// Mitsubishi GX Works2 project: FRA 451 Class Project   PLC: FX3G

PROGRAM MAIN
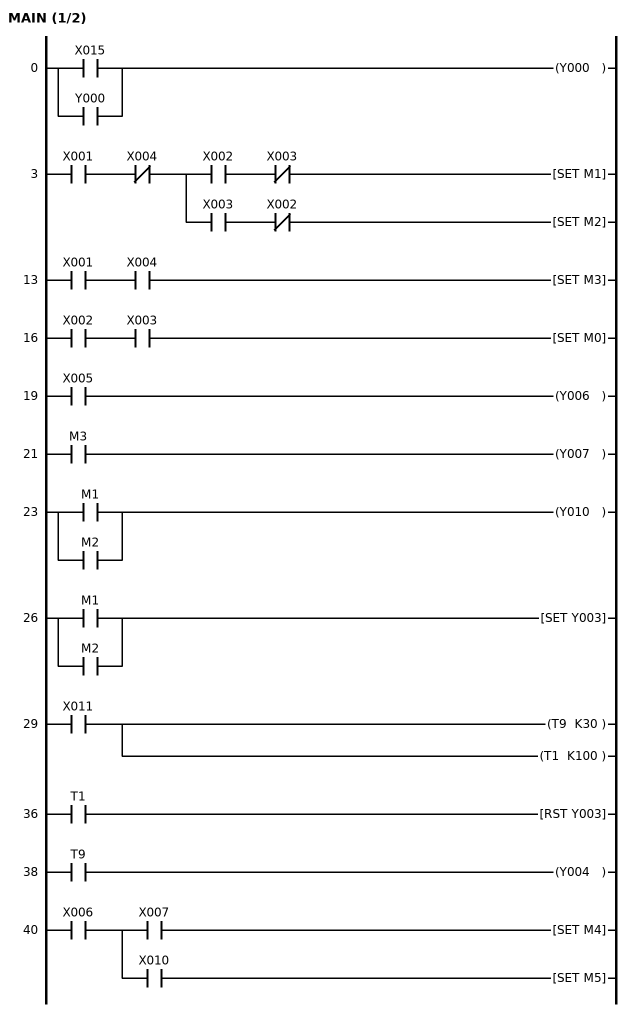
0     LD      X015
      OR      Y000
      OUT     Y000
3     LD      X001
      ANI     X004
      MPS
      AND     X002
      ANI     X003
      SET     M1
      MPP
      AND     X003
      ANI     X002
      SET     M2
13    LD      X001
      AND     X004
      SET     M3
16    LD      X002
      AND     X003
      SET     M0
19    LD      X005
      OUT     Y006
21    LD      M3
      OUT     Y007
23    LD      M1
      OR      M2
      OUT     Y010
26    LD      M1
      OR      M2
      SET     Y003
29    LD      X011
      OUT     T9 K30
      OUT     T1 K100
36    LD      T1
      RST     Y003
38    LD      T9
      OUT     Y004
40    LD      X006
      MPS
      AND     X007
      SET     M4
      MPP
      AND     X010
      SET     M5
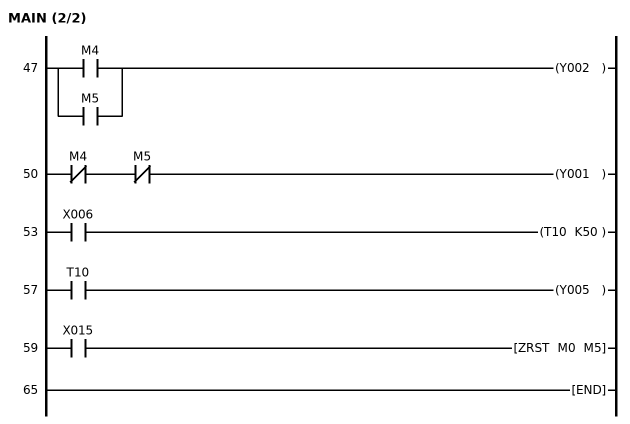
47    LD      M4
      OR      M5
      OUT     Y002
50    LDI     M4
      ANI     M5
      OUT     Y001
53    LD      X006
      OUT     T10 K50
57    LD      T10
      OUT     Y005
59    LD      X015
      ZRST    M0 M5
65    END
END_PROGRAM
